FUNCTION_BLOCK FB_InOnOff
VAR
	//Properties
	bError 				: BOOL 				:= FALSE;

	//value
	bValueIn			: BOOL;

	//Raw value
	bValueInRaw			AT %I* : BOOL;
END_VAR

PROPERTY Error : BOOL
GET
Error := THIS^.bError;
END_GET
SET
THIS^.bError := Error;
END_SET
END_PROPERTY

METHOD Read
bValueIn := bValueInRaw;
END_METHOD

PROPERTY ValueIn : BOOL
GET
ValueIn := THIS^.bValueIn;
END_GET
SET
THIS^.bValueIn := ValueIn;
END_SET
END_PROPERTY

END_FUNCTION_BLOCK

(* stored: Version 1.1.0.1, ProductVersion 3.1.4024.3
   POU FB_InOnOff: Id {67e160cd-5a71-4a38-950b-a6bd10bc48ca}, SpecialFunc None
   Property Error: Id {1be92a6d-0ba8-483f-92e2-0da30d228ff4}
   Get Get: Id {d7cdb247-bdb8-4dc9-af54-69106716b17c}
   Set Set: Id {f81c76bf-f9d8-4f30-851d-1863bdf30d30}
   Method Read: Id {3b68c215-86f0-49de-8d85-6a780fc756a2}
   Property ValueIn: Id {4832e14f-f1e0-449c-9239-7e9fecafff4d}
   Get Get: Id {75435d00-565f-41de-acbe-1ad45738a3e7}
   Set Set: Id {48077b17-3827-417a-8238-a9ae99629d9b} *)
